PROGRAM PRG_TEST
VAR
	fbDummyModule : FB_DummyModule;
END_VAR

(*
CONTAINS CODE NEEDED FOR AUTOMATIC TESTING
*)

// SystemBase is the master program. it controls all underlying modules.
SystemBase();

// Call modules
fbDummyModule(nModuleID:= 1);

// HMI control
// GVL_HMI.fbHMIControl();

END_PROGRAM

(* stored: Version 1.1.0.1, ProductVersion 3.1.4024.11
   POU PRG_TEST: Id {8fd80737-52d7-48f7-8910-0003a883abff}, SpecialFunc None *)
